PROGRAM TESTPRG
VAR
	// Currently there are no tests, except instantiating FUBs to make sure they build
	base : ComponentBase;
	runner : PluginRunner;
	taskBaseExtended : TaskBase;
END_VAR

TcUnit.RUN();

END_PROGRAM

(* stored: Version 1.1.0.1
   POU TESTPRG: Id {a9c53689-54d0-0ab2-03ea-b352bcf63e11}, SpecialFunc None *)
